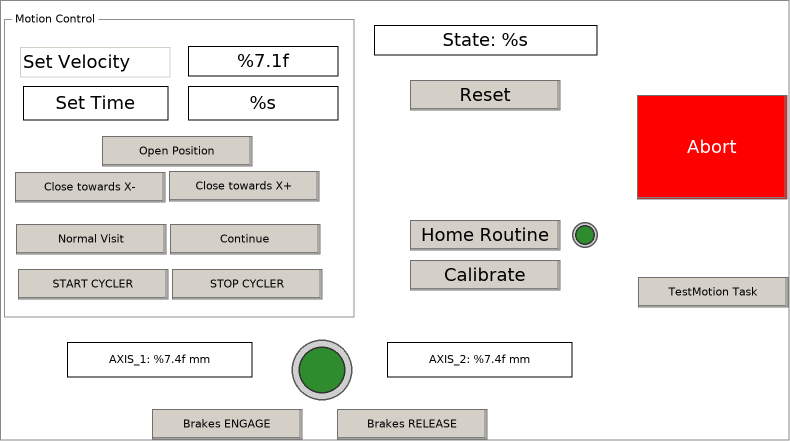
VISUALIZATION TestMotionGUI  // 790x441
    GroupBox (4,11 350x306), "Motion Control"
        Rectangle (19,75 145x34), "Set Time"
            OnMouseUp: write GVL.expoTime via Edit, min T#0.9s, format %7.1f
        Rectangle (184,75 150x34), "%s", text variable: GVL.expoTime
        Button (14,258 150x30), "START CYCLER", input disabled if: MAIN.testMotion.state <> 100;
            OnMouseUp: execute { MAIN.testMotionState:=3100; }
    Button (152,409 150x30), "Brakes ENGAGE"
        OnMouseClick: execute { GVL.brakeRelays := 0; }
    Button (337,409 150x30), "Brakes RELEASE"
        OnMouseClick: execute { GVL.brakeRelays := 3; }
    Lamp1 (287,335 70x70), variable: GVL.brakeRelays = 3, style: Lamp-Lamp1-Green
    Rectangle (67,342 185x35), "AXIS_1: %7.4f mm", text variable: MAIN.physicalAxes[0].NcToPlc.ActPos
    Rectangle (387,342 185x35), "AXIS_2: %7.4f mm", text variable: MAIN.physicalAxes[1].NcToPlc.ActPos
    Button (638,277 150x30), "TestMotion Task", input disabled if: GVL.task=2;
        OnMouseUp: execute { GVL.task:=2; }
    Button (410,80 150x30), "Reset"
        OnMouseUp: execute { MAIN.reset := TRUE; }
    Button (637,95 150x104), "Abort"
        OnMouseUp: execute { MAIN.abort := TRUE; }
    Rectangle (374,25 223x30), "State: %s", text variable: MAIN.testMotion.state;
    Button (410,220 150x30), "Home Routine", input disabled if: MAIN.testMotion.state <> 100;
        OnMouseUp: execute { MAIN.home := 3; }
    Button (102,136 150x30), "Open Position", input disabled if: MAIN.testMotion.state <> 100;
        OnMouseUp: execute { MAIN.testMotionState:=1000; }
    Textfield (20,47 150x30), "Set Velocity", input disabled if: MAIN.cycler.state <> ShutterState.STOPPED
        OnMouseUp: write MAIN.speed via Default, min 0, max 2000, format %7.1f
    Rectangle (188,46 150x30), "%7.1f", text variable: MAIN.speed
    Button (169,171 150x30), "Close towards X+", input disabled if: MAIN.testMotion.state <> 100;
        OnMouseUp: execute { MAIN.testMotionState:=1100; }
    Button (15,172 150x30), "Close towards X-", input disabled if: MAIN.testMotion.state <> 100;
        OnMouseUp: execute { MAIN.testMotionState:=1200; }
    Button (16,224 150x30), "Normal Visit", input disabled if: MAIN.testMotion.state <> 100;
        OnMouseUp: execute { MAIN.testMotionState:=2000; }
    Button (170,224 150x30), "Continue", input disabled if: MAIN.nextInstruct
        OnMouseUp: execute { MAIN.nextInstruct:=TRUE; }
    Lamp1 (570,220 30x30), variable: MAIN.physicalAxes[0].Status.Homed and MAIN.physicalAxes[1].Status.Homed;, style: Lamp-Lamp1-Green
    Button (410,260 150x30), "Calibrate", input disabled if: MAIN.testMotion.state <> 100;
        OnMouseUp: execute { MAIN.testMotionState:=9000; }
    Button (172,269 150x30), "STOP CYCLER"
        OnMouseUp: execute { MAIN.stop:=TRUE; }
END_VISUALIZATION

(* stored: Version 1.1.0.1, ProductVersion 3.1.4020.12
   Visu TestMotionGUI: Id {623b2af7-4d31-4390-b4d9-d32c32e32a74} *)
